TYPE ST_DataLog :
STRUCT
	sName:STRING;
	sName1:STRING;
	sName2:STRING;
	sName3:STRING;
	sName4:STRING;
	sValue:STRING;
END_STRUCT
END_TYPE

(* stored: Version 1.1.0.1, ProductVersion 3.1.4024.12
   DUT ST_DataLog: Id {ab76161f-2f79-484c-9d32-8bf82c49c2b1} *)
